(* IEC 61131-3 sources: mixture-prepar-plant/ST_code, 9 files *)

(* ---- AtmA.st ---- *)
FUNCTION_BLOCK PUBLIC AtmA EXTENDS Automaton
VAR_OUTPUT
    out: OutputA;
END_VAR
VAR
    tr_1_2: BOOL := FALSE;
    tr_2_3: BOOL := FALSE;
    tr_2_5: BOOL := FALSE;
    tr_3_4: BOOL := FALSE;
    tr_3_6: BOOL := FALSE;
    tr_4_1: BOOL := FALSE;
    tr_5_1: BOOL := FALSE;
    tr_6_1: BOOL := FALSE;
END_VAR

METHOD PRIVATE del : UINT
VAR_INPUT
    start:           BOOL := FALSE;
    ready:           BOOL := FALSE;
    reagentReady:    BOOL := FALSE;
    mixtureReady:    BOOL := FALSE;
    reagentSpoiled:  BOOL := FALSE;
    empty:           BOOL := FALSE;
    ackInterrupt:    BOOL := FALSE;
    mixtureDisposed: BOOL := FALSE;
END_VAR
VAR
    result: UINT;
END_VAR
BEGIN
    (* update transitions *)
    tr_1_2 := start AND ready;
    tr_2_3 := reagentReady AND NOT reagentSpoiled;
    tr_2_5 := reagentSpoiled;
    tr_3_4 := mixtureReady;
    tr_3_6 := reagentSpoiled AND NOT mixtureReady;
    tr_4_1 := empty;
    tr_5_1 := ackInterrupt;
    tr_6_1 := mixtureDisposed AND ackInterrupt;

    result := state;

    CASE state OF
        1:  IF    tr_1_2 THEN result := 2; END_IF
        2:  IF    tr_2_3 THEN result := 3;
            ELSIF tr_2_5 THEN result := 5; END_IF
        3:  IF    tr_3_4 THEN result := 4;
            ELSIF tr_3_6 THEN result := 6; END_IF
        4:  IF    tr_4_1 THEN result := 1; END_IF
        5:  IF    tr_5_1 THEN result := 1; END_IF
        6:  IF    tr_6_1 THEN result := 1; END_IF
    END_CASE

    del := result;
END

METHOD PRIVATE lam : OutputA
VAR_INPUT
    state: UINT;
END_VAR
BEGIN
    lam.preparingReagentIndicator := (state = 2);
    lam.preparingMixtureIndicator := (state = 3);
    lam.usingMixtureIndicator     := (state = 4);
    lam.interruptIndicator        := (state = 5) OR (state = 6);

    lam.prepareReagent     := (oldState = 1 AND tr_1_2);
    lam.prepareMixture     := (oldState = 2 AND tr_2_3);
    lam.stopPrepareMixture := (oldState = 3 AND tr_3_6) OR (oldState = 4 AND tr_4_1);

    lam.outletPump        := (state = 4);
    lam.mixtureValve      := (state = 4);
    lam.utilMixture       := (oldState = 3 AND tr_3_6);
    lam.initAfterDisposed := (oldState = 6 AND tr_6_1);
END

TYPE OutputA :
STRUCT
    preparingReagentIndicator: BOOL := FALSE;
    preparingMixtureIndicator: BOOL := FALSE;
    usingMixtureIndicator:     BOOL := FALSE;
    interruptIndicator:        BOOL := FALSE;
    prepareReagent:            BOOL := FALSE;
    prepareMixture:            BOOL := FALSE;
    stopPrepareMixture:        BOOL := FALSE;
    outletPump:                BOOL := FALSE;
    mixtureValve:              BOOL := FALSE;
    utilMixture:               BOOL := FALSE;
    initAfterDisposed:         BOOL := FALSE;
END_STRUCT
END_TYPE

METHOD PUBLIC iter
VAR_INPUT
    start:           BOOL := FALSE;
    ready:           BOOL := FALSE;
    reagentReady:    BOOL := FALSE;
    mixtureReady:    BOOL := FALSE;
    reagentSpoiled:  BOOL := FALSE;
    empty:           BOOL := FALSE;
    ackInterrupt:    BOOL := FALSE;
    mixtureDisposed: BOOL := FALSE;
END_VAR
BEGIN
    state := del(start, ready, reagentReady, mixtureReady, reagentSpoiled, empty, ackInterrupt, mixtureDisposed);
    out := lam(state);
    oldState := state;
END

END_FUNCTION_BLOCK

(* ---- AtmB.st ---- *)
FUNCTION_BLOCK PUBLIC AtmB EXTENDS Automaton
VAR_OUTPUT
    out: OutputB;
END_VAR
VAR
    tr_1_2: BOOL := FALSE;
    tr_2_3: BOOL := FALSE;
    tr_3_4: BOOL := FALSE;

    tr_2_1: BOOL := FALSE;
    tr_3_1: BOOL := FALSE;
    tr_4_1: BOOL := FALSE;
END_VAR

METHOD PRIVATE del : UINT
VAR_INPUT
    start:        BOOL := FALSE;
    reset:        BOOL := FALSE;
    high:         BOOL := FALSE;
    reagentAdded: BOOL := FALSE;
END_VAR
VAR
    result: UINT;
END_VAR
BEGIN
    (* update transitions *)
    tr_1_2 := start AND NOT reset;
    tr_2_3 := high AND NOT reset;
    tr_3_4 := reagentAdded AND NOT reset;
    tr_2_1 := reset;
    tr_3_1 := reset;
    tr_4_1 := reset;

    result := state;

    CASE state OF
        1:  IF    tr_1_2 THEN result := 2; END_IF
        2:  IF    tr_2_1 THEN result := 1;
            ELSIF tr_2_3 THEN result := 3; END_IF
        3:  IF    tr_3_1 THEN result := 1;
            ELSIF tr_3_4 THEN result := 4; END_IF
        4:  IF    tr_4_1 THEN result := 1; END_IF
    END_CASE

    del := result;
END

METHOD PRIVATE lam : OutputB
VAR_INPUT
    state: UINT;
    reset: BOOL;
END_VAR
BEGIN
    lam.waterValve  := (state = 2);
    lam.mixer       := (state = 3);
    lam.end         := (state = 4);
    lam.reagentFeed := (oldState = 2) AND tr_2_3;
    lam.resetSlave  := reset;
END

TYPE OutputB :
STRUCT
    waterValve:  BOOL := FALSE;
    mixer:       BOOL := FALSE;
    end:         BOOL := FALSE;
    reagentFeed: BOOL := FALSE;
    resetSlave:  BOOL := FALSE;
END_STRUCT
END_TYPE

METHOD PUBLIC iter
VAR_INPUT
    start:        BOOL := FALSE;
    reset:        BOOL := FALSE;
    high:         BOOL := FALSE;
    reagentAdded: BOOL := FALSE;
END_VAR
BEGIN
    state := del(start, reset, high, reagentAdded);
    out := lam(state, reset);
    oldState := state;
END

METHOD PUBLIC getEndPerspective : BOOL
VAR_INPUT
    start:        BOOL := FALSE;
    reset:        BOOL := FALSE;
    high:         BOOL := FALSE;
    reagentAdded: BOOL := FALSE;
END_VAR
VAR
    newState: UINT;
    newOut: OutputB;
END_VAR
BEGIN
    newState := del(start, reset, high, reagentAdded);
    newOut := lam(newState, reset);
    getEndPerspective := newOut.end;
END

END_FUNCTION_BLOCK

(* ---- AtmC.st ---- *)
FUNCTION_BLOCK PUBLIC AtmC EXTENDS Automaton
VAR_OUTPUT
    out: OutputC;
END_VAR
VAR
    tr_1_2:   BOOL := FALSE;
    tr_2_3:   BOOL := FALSE;
    tr_2_3_a: BOOL := FALSE;
    tr_2_3_b: BOOL := FALSE;
    tr_3_3:   BOOL := FALSE;
    tr_3_3_a: BOOL := FALSE;
    tr_3_3_b: BOOL := FALSE;
    tr_3_4:   BOOL := FALSE;
    tr_4_5:   BOOL := FALSE;

    tr_2_1:   BOOL := FALSE;
    tr_3_1:   BOOL := FALSE;
    tr_4_1:   BOOL := FALSE;
    tr_5_1:   BOOL := FALSE;
END_VAR

METHOD PRIVATE del : UINT
VAR_INPUT
    start:              BOOL := FALSE;
    pause:              BOOL := FALSE;
    reset:              BOOL := FALSE;
    reagentValveOpened: BOOL := FALSE;
    reagentValveClosed: BOOL := FALSE;
    full:               BOOL := FALSE;
END_VAR
VAR
    result: UINT;
END_VAR
BEGIN
    (* update transitions *)
    tr_1_2   := start AND NOT reset;
    tr_2_3_a := reagentValveOpened AND     pause AND NOT reset;
    tr_2_3_b := reagentValveOpened AND NOT pause AND NOT reset;
    tr_2_3   := tr_2_3_a OR tr_2_3_b;
    tr_3_3_a :=     pause AND NOT full AND NOT reset;
    tr_3_3_b := NOT pause AND NOT full AND NOT reset;
    tr_3_3   := tr_3_3_a OR tr_3_3_b;
    tr_3_4   := full AND NOT reset;
    tr_4_5   := reagentValveClosed AND NOT reset;

    tr_2_1 := reset;
    tr_3_1 := reset;
    tr_4_1 := reset;
    tr_5_1 := reset;

    result := state;

    CASE state OF
        1:  IF    tr_1_2 THEN result := 2; END_IF
        2:  IF    tr_2_1 THEN result := 1;
            ELSIF tr_2_3 THEN result := 3; END_IF
        3:  IF    tr_3_1 THEN result := 1;
            ELSIF tr_3_3 THEN result := 3;
            ELSIF tr_3_4 THEN result := 4; END_IF
        4:  IF    tr_4_1 THEN result := 1;
            ELSIF tr_4_5 THEN result := 5; END_IF
        5:  IF    tr_5_1 THEN result := 1; END_IF
    END_CASE

    del := result;
END

METHOD PRIVATE lam : OutputC
VAR_INPUT
    state: UINT;
END_VAR
BEGIN
    lam.reagentValveOpen  := (state = 2);
    lam.reagentValveClose := (state = 4);
    lam.end               := (state = 5);

    lam.inletPump := (oldState = 2 AND tr_2_3_b) OR
                     (oldState = 3 AND tr_3_3_b);
END

TYPE OutputC :
STRUCT
    reagentValveOpen:  BOOL := FALSE;
    reagentValveClose: BOOL := FALSE;
    inletPump:         BOOL := FALSE;
    end:               BOOL := FALSE;
END_STRUCT
END_TYPE

METHOD PUBLIC iter
VAR_INPUT
    start:              BOOL := FALSE;
    pause:              BOOL := FALSE;
    reset:              BOOL := FALSE;
    reagentValveOpened: BOOL := FALSE;
    reagentValveClosed: BOOL := FALSE;
    full:               BOOL := FALSE;
END_VAR
BEGIN
    state := del(start, pause, reset, reagentValveOpened, reagentValveClosed, full);
    out := lam(state);
    oldState := state;
END

METHOD PUBLIC getEndPerspective : BOOL
VAR_INPUT
    start:              BOOL := FALSE;
    pause:              BOOL := FALSE;
    reset:              BOOL := FALSE;
    reagentValveOpened: BOOL := FALSE;
    reagentValveClosed: BOOL := FALSE;
    full:               BOOL := FALSE;
END_VAR
VAR
    newState: UINT;
    newOut: OutputC;
END_VAR
BEGIN
    newState := del(start, pause, reset, reagentValveOpened, reagentValveClosed, full);
    newOut := lam(newState);
    getEndPerspective := newOut.end;
END

END_FUNCTION_BLOCK

(* ---- AtmD.st ---- *)
FUNCTION_BLOCK PUBLIC AtmD EXTENDS Automaton
VAR_OUTPUT
    out: OutputD;
END_VAR
VAR
    tr_1_2: BOOL := FALSE;
    tr_2_3: BOOL := FALSE;
    tr_3_4: BOOL := FALSE;
    tr_4_1: BOOL := FALSE;
    tr_4_5: BOOL := FALSE;
    tr_5_1: BOOL := FALSE;
END_VAR

METHOD PRIVATE del : UINT
VAR_INPUT
    start:             BOOL := FALSE;
    materialLoaded:    BOOL := FALSE;
    concentratePoured: BOOL := FALSE;
    homogenComplete:   BOOL := FALSE;
    reagentSpoiled:    BOOL := FALSE;
END_VAR
VAR
    result: UINT;
END_VAR
BEGIN
    (* update transitions *)
    tr_1_2 := start;
    tr_2_3 := materialLoaded;
    tr_3_4 := concentratePoured;
    tr_4_1 := reagentSpoiled;
    tr_4_5 := homogenComplete AND NOT reagentSpoiled;
    tr_5_1 := TRUE;

    result := state;

    CASE state OF
        1:  IF    tr_1_2 THEN result := 2; END_IF
        2:  IF    tr_2_3 THEN result := 3; END_IF
        3:  IF    tr_3_4 THEN result := 4; END_IF
        4:  IF    tr_4_1 THEN result := 1;
            ELSIF tr_4_5 THEN result := 5; END_IF
        5:  IF    tr_5_1 THEN result := 1; END_IF
    END_CASE

    del := result;
END

METHOD PRIVATE lam : OutputD
VAR_INPUT
    state: UINT;
END_VAR
BEGIN
    lam.startReagentStabilization := (oldState = 3 AND tr_3_4);

    lam.end := (state = 5);
END

TYPE OutputD :
STRUCT
    startReagentStabilization: BOOL := FALSE;
    end:                       BOOL := FALSE;
END_STRUCT
END_TYPE

METHOD PUBLIC iter
VAR_INPUT
    start:             BOOL := FALSE;
    materialLoaded:    BOOL := FALSE;
    concentratePoured: BOOL := FALSE;
    homogenComplete:   BOOL := FALSE;
    reagentSpoiled:    BOOL := FALSE;
END_VAR
BEGIN
    state := del(start, materialLoaded, concentratePoured, homogenComplete, reagentSpoiled);
    out := lam(state);
    oldState := state;
END

METHOD PUBLIC getEndPerspective : BOOL
VAR_INPUT
    start:             BOOL := FALSE;
    materialLoaded:    BOOL := FALSE;
    concentratePoured: BOOL := FALSE;
    homogenComplete:   BOOL := FALSE;
    reagentSpoiled:    BOOL := FALSE;
END_VAR
VAR
    newState: UINT;
    newOut: OutputD;
END_VAR
BEGIN
    newState := del(start, materialLoaded, concentratePoured, homogenComplete, reagentSpoiled);
    newOut := lam(newState);
    getEndPerspective := newOut.end;
END

END_FUNCTION_BLOCK

(* ---- AtmE.st ---- *)
FUNCTION_BLOCK PUBLIC AtmE EXTENDS Automaton
VAR_OUTPUT
    out: OutputE;
END_VAR
VAR
    tr_1_2:   BOOL := FALSE;
    tr_2_3:   BOOL := FALSE;
    tr_2_3_a: BOOL := FALSE;
    tr_2_3_b: BOOL := FALSE;
    tr_3_1:   BOOL := FALSE;
END_VAR

METHOD PRIVATE del : UINT
VAR_INPUT
    startStabil:     BOOL := FALSE;
    startUtil:       BOOL := FALSE;
    violated:        BOOL := FALSE;
    unstabilReagent: BOOL := FALSE;
    utilEnded:       BOOL := FALSE;
END_VAR
VAR
    result: UINT;
END_VAR
BEGIN
    (* update transitions *)
    tr_1_2   := startStabil;
    tr_2_3_a := startUtil;
    tr_2_3_b := violated AND NOT startUtil;
    tr_2_3   := tr_2_3_a OR tr_2_3_b;
    tr_3_1   := utilEnded;

    result := state;

    CASE state OF
        1:  IF tr_1_2 THEN result := 2; END_IF
        2:  IF tr_2_3 THEN result := 3; END_IF
        3:  IF tr_3_1 THEN result := 1; END_IF
    END_CASE

    del := result;
END

METHOD PRIVATE lam : OutputE
VAR_INPUT
    state: UINT;
    unstabilReagent: BOOL := FALSE;
END_VAR
BEGIN
    lam.unstabilReagent := (state = 2 AND unstabilReagent);
    lam.reagentSpoiled  := (oldState = 2 AND tr_2_3_b);
    lam.waiting         := (state = 1);
END

TYPE OutputE :
STRUCT
    unstabilReagent: BOOL := FALSE;
    reagentSpoiled:  BOOL := FALSE;
    waiting:         BOOL := TRUE;
END_STRUCT
END_TYPE

METHOD PUBLIC iter
VAR_INPUT
    startStabil:     BOOL := FALSE;
    startUtil:       BOOL := FALSE;
    violated:        BOOL := FALSE;
    unstabilReagent: BOOL := FALSE;
    utilEnded:       BOOL := FALSE;
END_VAR
BEGIN
    state := del(startStabil, startUtil, violated, unstabilReagent, utilEnded);
    out := lam(state, unstabilReagent);
    oldState := state;
END

METHOD PUBLIC getReagentSpoiledPerspective : BOOL
VAR_INPUT
    startStabil:     BOOL := FALSE;
    startUtil:       BOOL := FALSE;
    violated:        BOOL := FALSE;
    unstabilReagent: BOOL := FALSE;
    utilEnded:       BOOL := FALSE;
END_VAR
VAR
    newState: UINT;
    newOut: OutputE;
END_VAR
BEGIN
    newState := del(startStabil, startUtil, violated, unstabilReagent, utilEnded);
    newOut := lam(newState, unstabilReagent);
    getReagentSpoiledPerspective := newOut.reagentSpoiled;
END

END_FUNCTION_BLOCK

(* ---- AtmF.st ---- *)
FUNCTION_BLOCK PUBLIC AtmF EXTENDS Automaton
VAR_INPUT
    out: OutputF;
END_VAR
VAR_OUTPUT
END_VAR
VAR
    tr_1_2: BOOL := FALSE;
    tr_2_3: BOOL := FALSE;
    tr_3_4: BOOL := FALSE;
    tr_4_1: BOOL := FALSE;
END_VAR

METHOD PRIVATE del : UINT
VAR_INPUT
    start:              BOOL := FALSE;
    init:               BOOL := FALSE;
    empty:              BOOL := FALSE;
    reagentValveClosed: BOOL := FALSE;
END_VAR
VAR
    result: UINT;
END_VAR
BEGIN
    (* update transitions *)
    tr_1_2 := start;
    tr_2_3 := empty;
    tr_3_4 := reagentValveClosed;
    tr_4_1 := init;

    result := state;

    CASE state OF
        1:  IF tr_1_2 THEN result := 2; END_IF
        2:  IF tr_2_3 THEN result := 3; END_IF
        3:  IF tr_3_4 THEN result := 4; END_IF
        4:  IF tr_4_1 THEN result := 1; END_IF
    END_CASE

    del := result;
END

METHOD PRIVATE lam : OutputF
VAR_INPUT
    state: UINT;
END_VAR
BEGIN
    lam.outletPump        := (state = 2);
    lam.reagentValveClose := (state = 3);
    lam.end               := (state = 4);
END

TYPE OutputF :
STRUCT
    outletPump:        BOOL := FALSE;
    reagentValveClose: BOOL := FALSE;
    end:               BOOL := FALSE;
END_STRUCT
END_TYPE

METHOD PUBLIC iter
VAR_INPUT
    start:              BOOL := FALSE;
    init:               BOOL := FALSE;
    empty:              BOOL := FALSE;
    reagentValveClosed: BOOL := FALSE;
END_VAR
BEGIN
    state := del(start, init, empty, reagentValveClosed);
    out := lam(state);
    oldState := state;
END

END_FUNCTION_BLOCK

(* ---- Automaton.st ---- *)
FUNCTION_BLOCK PUBLIC Automaton
VAR
    state:    UINT := 1;
    oldState: UINT := state;
END_VAR

METHOD PUBLIC getState : UINT
BEGIN
    getState := state;
END

END_FUNCTION_BLOCK

(* ---- ControlModel.st ---- *)
FUNCTION_BLOCK PUBLIC ControlModel
VAR_OUTPUT
    out: OutputModel;
END_VAR
VAR
    atmA: AtmA;
    atmB: AtmB;
    atmC: AtmC;
    atmD: AtmD;
    atmE: AtmE;
    atmF: AtmF;

    atmE_waitingRetro: BOOL := FALSE;
    atmF_endRetro:     BOOL := FALSE;

    atmB_endPersp: BOOL := FALSE;
    atmC_endPersp: BOOL := FALSE;
    atmD_endPersp: BOOL := FALSE;
    atmE_reagentSpoiledPersp: BOOL := FALSE;
END_VAR

METHOD PUBLIC iter
VAR_INPUT
    start:              BOOL := FALSE;
    ackInterrupt:       BOOL := FALSE;
    full:               BOOL := FALSE;
    high:               BOOL := FALSE;
    empty:              BOOL := TRUE;
    reagentValveOpened: BOOL := FALSE;
    reagentValveClosed: BOOL := TRUE;
    materialLoaded:     BOOL := FALSE;
    concentratePoured:  BOOL := FALSE;
    homogenComplete:    BOOL := FALSE;
    violated:           BOOL := FALSE;
    unstabilReagent:    BOOL := FALSE;
    utilEnded:          BOOL := FALSE;
END_VAR
BEGIN
    (* Retrospectives *)
    atmE_waitingRetro := atmE.out.waiting;
    atmF_endRetro     := atmF.out.end;

    (* Perspectives *)
    atmC_endPersp := atmC.getEndPerspective( start := FALSE,
                                             pause := FALSE,
                                             reset := FALSE,
                                             reagentValveOpened := reagentValveOpened,
                                             reagentValveClosed := reagentValveClosed,
                                             full := full );
    atmB_endPersp := atmB.getEndPerspective( start := FALSE,
                                             reset := FALSE,
                                             high := high,
                                             reagentAdded := atmC_endPersp );
    atmE_reagentSpoiledPersp := atmE.getReagentSpoiledPerspective( startStabil := FALSE,
                                                                   startUtil := atmB_endPersp,
                                                                   violated := violated,
                                                                   unstabilReagent := unstabilReagent,
                                                                   utilEnded := utilEnded );
    atmD_endPersp := atmD.getEndPerspective( start := FALSE,
                                             materialLoaded := materialLoaded,
                                             concentratePoured := concentratePoured,
                                             homogenComplete := homogenComplete,
                                             reagentSpoiled := atmE_reagentSpoiledPersp );

    (* Automaton A *)
    atmA.iter( start := start,
               ready := atmE_waitingRetro,
               reagentReady := atmD_endPersp,
               mixtureReady := atmB_endPersp,
               reagentSpoiled := atmE_reagentSpoiledPersp,
               empty := empty,
               ackInterrupt := ackInterrupt,
               mixtureDisposed := atmF_endRetro );

    (* Automaton D *)
    atmD.iter( start := atmA.out.prepareReagent,
               materialLoaded := materialLoaded,
               concentratePoured := concentratePoured,
               homogenComplete := homogenComplete,
               reagentSpoiled := atmE_reagentSpoiledPersp );

    (* Automaton E *)
    atmE.iter( startStabil := atmD.out.startReagentStabilization,
               startUtil := atmB_endPersp,
               violated := violated,
               unstabilReagent := unstabilReagent,
               utilEnded := utilEnded );

    (* Automaton B *)
    atmB.iter( start := atmA.out.prepareMixture,
               reset := atmA.out.stopPrepareMixture,
               high := high,
               reagentAdded := atmC_endPersp );

    (* Automaton C *)
    atmC.iter( start := atmB.out.reagentFeed,
               pause := atmE.out.unstabilReagent,
               reset := atmB.out.resetSlave,
               reagentValveOpened := reagentValveOpened,
               reagentValveClosed := reagentValveClosed,
               full := full );

    (* Automaton F *)
    atmF.iter( start := atmA.out.utilMixture,
               init := atmA.out.initAfterDisposed,
               empty := empty,
               reagentValveClosed := reagentValveClosed );

    updateOutputs();
END

METHOD PRIVATE updateOutputs
BEGIN
    out.preparingReagentIndicator := atmA.out.preparingReagentIndicator;
    out.preparingMixtureIndicator := atmA.out.preparingMixtureIndicator;
    out.usingMixtureIndicator     := atmA.out.usingMixtureIndicator;
    out.interruptIndicator        := atmA.out.interruptIndicator;

    out.waterValve   := atmB.out.waterValve;
    out.mixtureValve := atmA.out.mixtureValve;
    out.mixer        := atmB.out.mixer;

    out.reagentValveOpen  := atmC.out.reagentValveOpen;
    out.reagentValveClose := atmC.out.reagentValveClose OR atmF.out.reagentValveClose;
    out.inletPump         := atmC.out.inletPump;
    out.outletPump        := atmA.out.outletPump OR atmF.out.outletPump;
END

TYPE OutputModel :
STRUCT
    preparingReagentIndicator: BOOL := FALSE;
    preparingMixtureIndicator: BOOL := FALSE;
    usingMixtureIndicator:     BOOL := FALSE;
    interruptIndicator:        BOOL := FALSE;
    waterValve:                BOOL := FALSE;
    mixtureValve:              BOOL := FALSE;
    mixer:                     BOOL := FALSE;
    reagentValveOpen:          BOOL := FALSE;
    reagentValveClose:         BOOL := FALSE;
    inletPump:                 BOOL := FALSE;
    outletPump:                BOOL := FALSE;
END_STRUCT
END_TYPE

METHOD PUBLIC getState : ModelState
BEGIN
    getState.stateA := atmA.getState();
    getState.stateB := atmB.getState();
    getState.stateC := atmC.getState();
    getState.stateD := atmD.getState();
    getState.stateE := atmE.getState();
    getState.stateF := atmF.getState();
END

TYPE ModelState :
STRUCT
    stateA: UINT;
    stateB: UINT;
    stateC: UINT;
    stateD: UINT;
    stateE: UINT;
    stateF: UINT;
END_STRUCT
END_TYPE

END_FUNCTION_BLOCK

(* ---- PLC_PRG.st ---- *)
PROGRAM PLC_PRG
VAR
    model: ControlModel;
    state: ModelState;

    (* Inputs *)
    start:              BOOL := FALSE;
    ackInterrupt:       BOOL := FALSE;
    full:               BOOL := FALSE;
    high:               BOOL := FALSE;
    empty:              BOOL := TRUE;
    reagentValveOpened: BOOL := FALSE;
    reagentValveClosed: BOOL := TRUE;
    materialLoaded:     BOOL := FALSE;
    concentratePoured:  BOOL := FALSE;
    homogenComplete:    BOOL := FALSE;
    violated:           BOOL := FALSE;
    unstabilReagent:    BOOL := FALSE;
    utilEnded:          BOOL := FALSE;
END_VAR
BEGIN
    model.iter( start,
                ackInterrupt,
                full,
                high,
                empty,
                reagentValveOpened,
                reagentValveClosed,
                materialLoaded,
                concentratePoured,
                homogenComplete,
                violated,
                unstabilReagent,
                utilEnded );
    state := model.getState();
END_PROGRAM
